// TwinCAT 3 PLC project Main
// ProgramVersion: 3.1.4023.0
// libraries:
//   Tc2_Standard, * (Beckhoff Automation GmbH)
//   Tc2_System, * (Beckhoff Automation GmbH)
//   Tc3_Module, * (Beckhoff Automation GmbH)
// project tree:
//   DUTs/ StructureWithArray.TcDUT, StructureWithStructureWithArray.TcDUT
//   GVLs/ GVL.TcGVL
//   / PlcTask.TcTTO
//   POUs/ MAIN.TcPOU
// real-time tasks:
//   TASK PlcTask: cycle T#10ms, priority 20, ADS port 350

CONFIGURATION Main
    RESOURCE PLC ON TwinCAT3
        TASK PlcTask(INTERVAL := T#10ms, PRIORITY := 20);
        PROGRAM MAIN WITH PlcTask : MAIN;
    END_RESOURCE
END_CONFIGURATION

// ---- DUTs/StructureWithArray.TcDUT
TYPE StructureWithArray :
STRUCT
	myArray : ARRAY [0..2] OF LREAL;
END_STRUCT
END_TYPE

// ---- DUTs/StructureWithStructureWithArray.TcDUT
TYPE StructureWithStructureWithArray :
STRUCT
	myStruct : StructureWithArray;
END_STRUCT
END_TYPE

// ---- GVLs/GVL.TcGVL
{attribute 'qualified_only'}
VAR_GLOBAL

	structureWithStructureWithArray : StructureWithStructureWithArray;
	structureWithArray : structureWithArray;
	
	arrayWithStructureWithArray : ARRAY [0..2] OF structureWithArray;

END_VAR

// ---- POUs/MAIN.TcPOU
PROGRAM MAIN
VAR
	values : ARRAY [0..24] OF LREAL;
	i : int;
END_VAR

values[0] := values[0] + 1;

IF values[0] > 100 THEN
	values[0] := 0;
END_IF

FOR i := 1 TO 24 DO
	values[i] := values[0] + (i * 10);
	
	gvl.arrayWithStructureWithArray[0].myArray[0] := values[0];
	gvl.structureWithArray.myArray[0] := values[0];
	gvl.structureWithStructureWithArray.myStruct.myArray[0] := values[0];
	
END_FOR

END_PROGRAM
